TYPE ST_highLevelCtrlSig :
STRUCT
	m_faultMask:ARRAY [1..g_sArmNum] OF BOOL:=[4(0)];
	
	
END_STRUCT
END_TYPE

(* stored: Version 1.1.0.1, ProductVersion 3.1.4024.11
   DUT ST_highLevelCtrlSig: Id {bef0044b-eb1e-43eb-9495-0bc1484501d6} *)
